{attribute 'qualified_only'}
VAR_GLOBAL CONSTANT
	MaxObservers 	: INT := 5;	
END_VAR

(* stored: Version 1.1.0.1, ProductVersion 3.1.4024.11
   GVL Param: Id {5105eb29-77e8-44b8-9f51-83fde952f942}, ParameterList True *)
